{attribute 'GeneratedUsingTerminal: EK1100-0000-0018'}
{attribute addProperty BoxType "EK1100-0000-0018"}
{attribute addProperty Id "Beckhoff_CXxxxxEK1122Beckhoff_CXxxxxEK1122_5A4CF81D176"}
{attribute addProperty CRC "3311340148"}
{attribute addProperty Size "176"}
TYPE Beckhoff_CXxxxx_C55F0A74 EXTENDS EK1100_1FC0878B :
STRUCT
	{attribute addProperty Name "Beckhoff_CXxxxxEK1122"}
	{attribute addProperty PreviousPort "Beckhoff CXxxxx : B"}
	Beckhoff_CXxxxxEK1122 : Beckhoff_CXxxxxEK1122_5A4CF81D;
END_STRUCT
END_TYPE

(* stored: Version 1.2.0.0, ProductVersion 3.1.4024.9
   DUT Beckhoff_CXxxxx_C55F0A74: Id {860a7fb4-c2e3-4be9-be65-38c917263801} *)
